// TIA Portal V19 export
TYPE "JB_Status"
   STRUCT
      Torch : "Positioning_DOL_Machine_COut";
      ClampEntry : "ValveMachine_COut";
      ClampExit : "ValveMachine_COut";
      CutHead : "ValveMachine_COut";
      Pinchroll_Feed : "SpeedMachine_COut";
      Pinchroll_Lift : "ValveMachine_COut";
      Cut_ManCycleDone : Bool;
      Weld_CheckNext : Bool;
      TorchInParkPosition : Bool;
      JunctionDone : Bool;
   END_STRUCT;
END_TYPE
